// TIA Portal V17 export
// export: Created 2023-05-07T12:12:09.1582926Z, ExportSetting WithDefaults, DisplayName Totally Integrated Automation Portal, DisplayVersion V17, DisplayName TIA Portal Openness, DisplayVersion V17, DisplayName TIA Portal Version Control Interface, DisplayVersion V17, DisplayName TIA Portal Test Suite Advanced, DisplayVersion V17, DisplayName STEP 7 Professional, DisplayVersion V17, DisplayName SIMATIC Energy Suite, DisplayVersion V17, DisplayName STEP 7 Safety, DisplayVersion V17, DisplayName WinCC Professional, DisplayVersion V17
ORGANIZATION_BLOCK "PID_C"   // OB30, LAD, CyclicInterrupt
{ S7_Optimized_Access := 'TRUE' }
VERSION : 0.1
// stored: AutoNumber true, IsIECCheckEnabled false, SetENOAutomatically false
   VAR_INPUT
      Initial_Call : Bool;   // Initial call of this OB
      Event_Count : Int;   // Events discarded
   END_VAR
BEGIN

REGION Network 1: PID_Compact
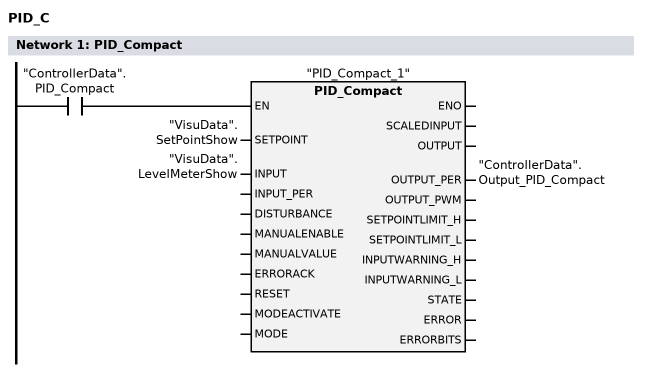
   RUNG wire#powerrail
      Contact( "ControllerData".PID_Compact )
      "PID_Compact_1".PID_Compact(Setpoint := "VisuData".SetPointShow, Input := "VisuData".LevelMeterShow, Input_PER :=, Disturbance :=, ManualEnable :=, ManualValue :=, ErrorAck :=, Reset :=, ModeActivate :=, Mode :=, ScaledInput =>, Output =>, Output_PER => "ControllerData".Output_PID_Compact, Output_PWM =>, SetpointLimit_H =>, SetpointLimit_L =>, InputWarning_H =>, InputWarning_L =>, State =>, Error =>, ErrorBits =>)
   END_RUNG
   // the same network as SCL:
   IF "ControllerData".PID_Compact THEN
       "PID_Compact_1"(Setpoint := "VisuData".SetPointShow,   // PID_Compact
                       Input := "VisuData".LevelMeterShow,
                       Output_PER => "ControllerData".Output_PID_Compact);
   END_IF;
END_REGION
END_ORGANIZATION_BLOCK
